ABB RAPID module: RoboData.mod

MODULE RoboData


    ! --- Tool and Work Objects ---
    TASK PERS tooldata tsuck:=[TRUE,[[-213.978,-32.7493,167.349],[1,0,0,0]],[1.1,[0,20,25],[1,0,0,0],0,0,0]];
    TASK PERS wobjdata wobj1:=[FALSE,TRUE,"",[[959.838,-291.657,795.046],[0.999978,-0.00504122,0.00423326,6.27363E-05]],[[0,0,0],[1,0,0,0]]];
    TASK PERS wobjdata wobjAiPlaceTray:=[FALSE,TRUE,"",[[1260.7,-295.297,805.883],[0.999907,0.00186707,-0.0135008,7.64184E-05]],[[0,0,0],[1,0,0,0]]];
    TASK PERS wobjdata wobjAruco:=[FALSE,TRUE,"",[[1190.74,291.064,795.822],[0.999893,-0.012889,-0.00608741,-0.00331874]],[[0,0,0],[1,0,0,0]]];

    ! --- Dynamic Target (updated by Python) ---
    PERS robtarget shape:=[[118.29,-181.05,2],[0.00826666,0.157305,-0.987506,-0.00431963],[0,0,-1,0],[9E+09,9E+09,9E+09,9E+09,9E+09,9E+09]];

    ! --- Static Place Targets ---
    CONST robtarget pHome:=[[197.51,429.20,349.54],[0.00855298,-0.546338,0.83751,0.00434769],[0,0,-1,0],[9E+09,9E+09,9E+09,9E+09,9E+09,9E+09]];
    CONST robtarget pApporach:=[[197.83,-7.46,305.10],[0.00855917,-0.546322,0.83752,0.00435965],[-1,0,-1,0],[9E+09,9E+09,9E+09,9E+09,9E+09,9E+09]];
    ! --- Tray placements for wobjs wobjAiPlaceTray
    CONST robtarget pCircle:=[[141.13,-72.22,184.39],[0.00845965,-0.54632,0.837522,0.00447932],[-1,0,-1,0],[9E+09,9E+09,9E+09,9E+09,9E+09,9E+09]];
    CONST robtarget pSquare:=[[152.08,58.50,186.68],[0.00844458,-0.546334,0.837513,0.00449096],[-1,0,-1,0],[9E+09,9E+09,9E+09,9E+09,9E+09,9E+09]];
    CONST robtarget pStar:=[[204.15,-4.80,187.79],[0.00844077,-0.546314,0.837526,0.00448595],[-1,0,-1,0],[9E+09,9E+09,9E+09,9E+09,9E+09,9E+09]];
    CONST robtarget pHexagon:=[[249.92,-64.96,186.22],[0.00844813,-0.546312,0.837527,0.00447767],[-1,0,-1,0],[9E+09,9E+09,9E+09,9E+09,9E+09,9E+09]];
    CONST robtarget pTriangle:=[[263.32,47.40,189.26],[0.00845512,-0.546317,0.837524,0.00446771],[-1,0,-1,0],[9E+09,9E+09,9E+09,9E+09,9E+09,9E+09]];



ENDMODULE
